// TIA Portal V20 export
DATA_BLOCK "CONTROL_ON_FB_IDB"   // DB30230
// stored: AssignedProDiagFB GENERAL_PD, AutoNumber false, InstanceOfName CONTROL_ON_OFF_PD_FB, InstanceOfType FB
"CONTROL_ON_OFF_PD_FB"
   // VAR_INPUT
   //    PLANT_IDENTIFIER { ExternalAccessible := 'False'; ExternalVisible := 'False'; ExternalWritable := 'False'} : WString[24];
   //    ENABLE_CONTROL_ON { ExternalAccessible := 'False'; ExternalVisible := 'False'; ExternalWritable := 'False'} : Bool;
   //    PUSHBUTTON_ON { ExternalAccessible := 'False'; ExternalVisible := 'False'; ExternalWritable := 'False'} : Bool;
   //    PUSHBUTTON_OFF { ExternalAccessible := 'False'; ExternalVisible := 'False'; ExternalWritable := 'False'} : Bool;
   //    CONTACTOR_FEEDBACK { ExternalAccessible := 'False'; ExternalVisible := 'False'; ExternalWritable := 'False'} : Bool;
   //    RESET { ExternalAccessible := 'False'; ExternalVisible := 'False'; ExternalWritable := 'False'} : Bool;
   //    TIME_FEEDBACK_ON { ExternalAccessible := 'False'; ExternalVisible := 'False'; ExternalWritable := 'False'} : Time;
   //    TIME_DELAY_1 { ExternalAccessible := 'False'; ExternalVisible := 'False'; ExternalWritable := 'False'} : Time;
   //    TIME_DELAY_2 { ExternalAccessible := 'False'; ExternalVisible := 'False'; ExternalWritable := 'False'} : Time;
   //    "GLOBAL_CLOCK&SYSTEM" { ExternalAccessible := 'False'; ExternalVisible := 'False'; ExternalWritable := 'False'} : "GLOBAL_CLOCK&SYSTEM_MEMORY_UDT";
   // END_VAR
   // VAR_OUTPUT
   //    GENERAL_ALARM { ExternalAccessible := 'False'; ExternalVisible := 'False'; ExternalWritable := 'False'} : Bool;
   //    CONTACTER_ON { ExternalAccessible := 'False'; ExternalVisible := 'False'; ExternalWritable := 'False'} : Bool;
   //    CONTROL_ON { ExternalAccessible := 'False'; ExternalVisible := 'False'; ExternalWritable := 'False'} : Bool;
   //    CONTROL_ON_DELAYED_1 { ExternalAccessible := 'False'; ExternalVisible := 'False'; ExternalWritable := 'False'} : Bool;
   //    CONTROL_ON_DELAYED_2 { ExternalAccessible := 'False'; ExternalVisible := 'False'; ExternalWritable := 'False'} : Bool;
   //    EXTENDED_PULSE_PLC_ON { ExternalAccessible := 'False'; ExternalVisible := 'False'; ExternalWritable := 'False'} : Bool;
   //    CONTROL_ON_DISPLAY { ExternalAccessible := 'False'; ExternalVisible := 'False'; ExternalWritable := 'False'} : Bool;
   //    CONTROL_OFF_DISPLAY { ExternalAccessible := 'False'; ExternalVisible := 'False'; ExternalWritable := 'False'} : Bool;
   // END_VAR
   // VAR
   //    HMI_IN : Byte;
   //    HMI_ON_OFF_Header : Byte;
   //    HMI_OFF : Byte;
   //    HMI_ON : Bool;
   //    HMI_Req_OFF : Bool;
   //    Instruction { ExternalAccessible := 'False'; ExternalVisible := 'False'; ExternalWritable := 'False'} : Struct
   //       Timer_Feedback_On { S7_SetPoint := 'True'} : IEC_TIMER;
   //       Timer_Control_ON_delay_1 { S7_SetPoint := 'True'} : IEC_TIMER;
   //       Timer_Control_ON_delay_2 { S7_SetPoint := 'True'} : IEC_TIMER;
   //       Timer_Control_ON_display { S7_SetPoint := 'True'} : IEC_TIMER;
   //       PLC_delay_ON { S7_SetPoint := 'True'} : IEC_TIMER;
   //       Extended_PLC_ON { S7_SetPoint := 'True'} : IEC_TIMER;
   //    END_STRUCT;
   //    Alarm { ExternalAccessible := 'False'; ExternalVisible := 'False'; ExternalWritable := 'False'} : Struct
   //       T_FeedBack_ON : Bool;
   //       FeedBack_Lost_no_cmd : Bool;
   //       Enable_missing : Bool;
   //       Spare_3 : Bool;
   //       Spare_4 : Bool;
   //       Spare_5 : Bool;
   //       Spare_6 : Bool;
   //       Spare_7 : Bool;
   //       Spare_8 : Bool;
   //       Spare_9 : Bool;
   //       Spare_10 : Bool;
   //       Spare_11 : Bool;
   //       Spare_12 : Bool;
   //       Spare_13 : Bool;
   //       Spare_14 : Bool;
   //       Spare_15 : Bool;
   //    END_STRUCT;
   //    PE { ExternalAccessible := 'False'; ExternalVisible := 'False'; ExternalWritable := 'False'} : Struct
   //       AlarmReset : Bool;
   //       ControlON : Bool;
   //       ControlOFF : Bool;
   //       ReqOFF : Bool;
   //    END_STRUCT;
   //    PP { ExternalAccessible := 'False'; ExternalVisible := 'False'; ExternalWritable := 'False'} : Struct
   //       AlarmReset : Bool;
   //       ControlON : Bool;
   //       ControlOFF : Bool;
   //       ReqOFF : Bool;
   //    END_STRUCT;
   //    NE { ExternalAccessible := 'False'; ExternalVisible := 'False'; ExternalWritable := 'False'} : Struct
   //       Feedback_On : Bool;
   //       ReqOFF : Bool;
   //       ControlOFF : Bool;
   //    END_STRUCT;
   //    NP { ExternalAccessible := 'False'; ExternalVisible := 'False'; ExternalWritable := 'False'} : Struct
   //       Feedback_On : Bool;
   //       ReqOFF : Bool;
   //       ControlOFF : Bool;
   //    END_STRUCT;
   //    AX { ExternalAccessible := 'False'; ExternalVisible := 'False'; ExternalWritable := 'False'} : Struct
   //       FirstCycle : Bool;
   //       ControlOFF_Req : Bool;
   //       ControlOFF_active : Bool;
   //       ContactorON : Bool;
   //       General_Alarm : Bool;
   //       Control_ON_delayed_1 : Bool;
   //       Control_ON_delayed_2 : Bool;
   //       Control_ON : Bool;
   //       Extended_PLC_ON : Bool;
   //       Control_ON_display : Bool;
   //    END_STRUCT;
   //    Alarm_No_PD { ExternalAccessible := 'False'; ExternalVisible := 'False'; ExternalWritable := 'False'} : UInt;
   //    GLOBAL_GENERAL_AlarmTextList_Item { ExternalAccessible := 'False'; ExternalVisible := 'False'; ExternalWritable := 'False'} : USInt;
   // END_VAR
BEGIN
END_DATA_BLOCK
